FUNCTION_BLOCK FB_Inventory
VAR_INPUT
END_VAR
VAR_OUTPUT
END_VAR
VAR
	_stInventory : ARRAY [0..5] OF ST_ProductInfo;
	_nNumberProducts : INT := 0;
	_fTotalWeight : REAL;
	_fTotalVolume : REAL;
END_VAR

METHOD FB_init : BOOL
VAR_INPUT
	bInitRetains : BOOL; // if TRUE, the retain variables are initialized (warm start / cold start)
	bInCopyCode : BOOL;  // if TRUE, the instance afterwards gets moved into the copy code (online change)
	product1 : ST_ProductInfo;
	product2 : ST_ProductInfo;
END_VAR
M_Add(product1);
M_Add(product2);
END_METHOD

PROPERTY PUBLIC fTotalVolume : REAL
GET
END_GET
SET
END_SET
END_PROPERTY

PROPERTY PUBLIC fTotalWeight : REAL
GET
END_GET
SET
END_SET
END_PROPERTY

METHOD PUBLIC M_Add
VAR_INPUT
	stProductInfo : ST_ProductInfo;
END_VAR
_stInventory[_nNumberProducts] := stProductInfo;
_nNumberProducts := _nNumberProducts + 1;
END_METHOD

METHOD PRIVATE M_CalculateVolume
VAR_INPUT
END_VAR
END_METHOD

METHOD PRIVATE M_CalculateWeight
VAR_INPUT
END_VAR
END_METHOD

METHOD PUBLIC M_Remove
VAR_INPUT
	nIndex : INT;
END_VAR
VAR
	stNullProduct : ST_ProductInfo := (eproductType := E_ProductType.cube, fDimension1 := 0, fDimension2 := 0, fDimension3 := 0, fSpecificWeight := 0);
END_VAR
_stInventory[nIndex] := _stInventory[_nNumberProducts - 1];
_stInventory[_nNumberProducts - 1] := stNullProduct;
_nNumberProducts := _nNumberProducts - 1;
END_METHOD

PROPERTY PUBLIC nNumberProducts : INT
GET
END_GET
SET
END_SET
END_PROPERTY

PROPERTY PUBLIC stInventory : array [1..5] of ST_ProductInfo
GET
END_GET
SET
END_SET
END_PROPERTY

END_FUNCTION_BLOCK

(* stored: Version 1.1.0.1, ProductVersion 3.1.4024.13
   POU FB_Inventory: Id {1590838d-79b5-42ab-a987-ea8205388890}, SpecialFunc None
   Method FB_init: Id {a3ca062b-5c77-4d2d-ad09-0a04b60bebd6}
   Property fTotalVolume: Id {2b8f90b8-98a7-47c5-8cdf-19bbe890623a}
   Get Get: Id {2bbdf9be-86a6-4871-b6f7-07eded515274}
   Set Set: Id {b86e48e7-18eb-4773-81d0-3b8eea87d0e6}
   Property fTotalWeight: Id {37f700be-56a1-4853-b670-b1b197d28c9f}
   Get Get: Id {cc6cadc8-9e33-4d76-87bc-7800bd309193}
   Set Set: Id {f5c8fff1-606e-4959-8c39-3eabed6040d7}
   Method M_Add: Id {60b6ffc1-062c-4858-a5b9-496d0cf9a5e1}
   Method M_CalculateVolume: Id {ca098987-d7c7-49fb-be5e-a714b879e2ce}
   Method M_CalculateWeight: Id {fc436bc6-3362-4a30-ab1f-e272faa93133}
   Method M_Remove: Id {d8764512-37aa-4b16-b675-337ad4ad0d0e}
   Property nNumberProducts: Id {edca9347-19db-4646-898e-439040ff7875}
   Get Get: Id {ba336513-34b5-40f1-a77c-aee2a36441fc}
   Set Set: Id {65b8b70c-f6cd-47e3-80fa-41ccde37ca22}
   Property stInventory: Id {5c5bfa9c-de03-4dc2-83b6-1d39960c8e07}
   Get Get: Id {c0dad690-bdb6-4d58-a3f7-4dfef74d5921}
   Set Set: Id {81453f42-ec0d-4f40-917f-6a1082e2e96e} *)
